FUNCTION_BLOCK Machine EXTENDS FB_PackML_BaseModule
VAR
	LeftPress  : Press := (Name := 'Left Press', GroupId := 0);	 //4. GroupId used to match up with AxisAssignment
	RightPress : Press := (Name := 'Right Press', GroupId := 1); //4. GroupId used to match up with AxisAssignment

	//
	AxisAssignment : ARRAY[1..GVL_AXES.MAX_AXES] OF INT;

	//
	HMI : ST_Machine_HMI;
END_VAR

(* This method contains code which will execute when this PackML module is in the Clearing state*)
METHOD PROTECTED Clearing
// 8.b. This will pass the radio button selections to each EM.
LeftPress.ActiveAxes  := AxisAssignment;
RightPress.ActiveAxes := AxisAssignment;

//
SUPER^.Clearing();
END_METHOD

METHOD CyclicLogic
IF NOT _InitComplete THEN
	_InitComplete := Initialize();
	RETURN;
END_IF

SUPER^.CyclicLogic();
END_METHOD

(* This method contains code which will execute when this PackML module is in the Execute state*)
METHOD PROTECTED Execute
CASE _CurrentMode OF
	E_PMLUnitMode.Production:
		IF HMI.Cmd.MoveAll THEN
			HMI.Cmd.MoveAll := FALSE;
			LeftPress.MoveAll(100.0);
			RightPress.MoveAll(-100.0);
		END_IF
END_CASE
END_METHOD

(* Automatically enables and disables HMI control based on the PackML mode*)
METHOD PROTECTED HMIPermissions
AllowHMIControl(TRUE);
END_METHOD

(* Basic module initialization logic*)
METHOD PROTECTED Initialize : BOOL
Initialize := FALSE;
CASE DescendantSequenceState OF
	0:
		RegisterSubmodule(SubModule := LeftPress);
		RegisterSubmodule(SubModule := RightPress);
		DescendantSequenceState := DescendantSequenceState + 10;

	10:
		IF SUPER^.Initialize() THEN
			DescendantSequenceState := DescendantSequenceState + 10;
		END_IF

	20:
		Initialize := TRUE;
END_CASE
END_METHOD

END_FUNCTION_BLOCK

(* stored: Version 1.1.0.1
   POU Machine: Id {8b1e344a-67f4-4ac0-acc9-f85d1bd9c057}, SpecialFunc None
   Folder Acting States: Id {dc272a52-cbda-4c9d-9bb4-d1778504f1bd}
   Folder CyclicLogic: Id {7dd02334-f591-4752-9bf4-7b719aade17c}
   Folder Initialize: Id {63354e98-63d6-4ba5-9878-a8ec70c17a07}
   Folder Waiting States: Id {165ef01e-3862-40dc-a9cd-c9c81cb74308}
   Method Clearing: Id {520ca38d-f422-408c-a0e6-b1e66da495b2}
   Method CyclicLogic: Id {f22d268b-ccea-498c-9d8f-56a8731d21aa}
   Method Execute: Id {1615e559-0337-4d00-8934-af1bba18f39c}
   Method HMIPermissions: Id {0f3a45a6-4cb0-4028-82cc-2e96d0c70c99}
   Method Initialize: Id {007542e4-7de5-4f40-a8e0-a816e4fa97a1} *)
